{attribute addProperty BoxType "EP9224-0037-0017"}
{attribute addProperty Id "Warning_TemperatureBIT10.1251Error_TemperatureBIT10.1252Warning_UsBIT10.1253Error_UsBIT10.1254Warning_UpBIT10.1255Error_UpBIT10.1256Global_Error_BitBIT10.1257Warning_Sum_CurrentBIT10.1258Error_Sum_CurrentBIT10.1259TxPDO_StateBIT10.12515TxPDO_ToggleBIT10.12516"}
{attribute addProperty CRC "1062916947"}
{attribute addProperty SizeInBites "16"}
{attribute addProperty SizeInBytes "2"}
TYPE Device_Status_3F5AD353 :
STRUCT
	{attribute addProperty Name "Warning_Temperature"}
	Warning_Temperature : BIT;
	{attribute addProperty Name "Error_Temperature"}
	Error_Temperature : BIT;
	{attribute addProperty Name "Warning_Us"}
	Warning_Us : BIT;
	{attribute addProperty Name "Error_Us"}
	Error_Us : BIT;
	{attribute addProperty Name "Warning_Up"}
	Warning_Up : BIT;
	{attribute addProperty Name "Error_Up"}
	Error_Up : BIT;
	{attribute addProperty Name "Global_Error_Bit"}
	Global_Error_Bit : BIT;
	{attribute addProperty Name "Warning_Sum_Current"}
	Warning_Sum_Current : BIT;
	{attribute addProperty Name "Error_Sum_Current"}
	Error_Sum_Current : BIT;
	{attribute 'hide'}
	reserve_1_BIT_0 : BIT;
	{attribute 'hide'}
	reserve_1_BIT_1 : BIT;
	{attribute 'hide'}
	reserve_1_BIT_2 : BIT;
	{attribute 'hide'}
	reserve_1_BIT_3 : BIT;
	{attribute 'hide'}
	reserve_1_BIT_4 : BIT;
	{attribute addProperty Name "TxPDO_State"}
	TxPDO_State : BIT;
	{attribute addProperty Name "TxPDO_Toggle"}
	TxPDO_Toggle : BIT;
END_STRUCT
END_TYPE

(* stored: Version 1.2.0.0, ProductVersion 3.1.4024.9
   DUT Device_Status_3F5AD353: Id {757ed32c-9d78-4864-a925-da4fe23686f6} *)
